TYPE ST_BaseHMIControlElement_Command_Link :
STRUCT
END_STRUCT
END_TYPE

(* stored: Version 1.1.0.1
   DUT ST_BaseHMIControlElement_Command_Link: Id {d7daf18e-34ad-026a-052d-a77acc0b6186} *)
